TYPE IoEd12dssShutter :
STRUCT	
	OutputSwitchContactClosure	AT %Q* : BOOL;	
	
	inputShutter1 AT %I* : BOOL;
	inputShutter2 AT %I* : BOOL;
END_STRUCT
END_TYPE

(* stored: Version 1.1.0.1, ProductVersion 3.1.4024.4
   DUT IoEd12dssShutter: Id {a2021377-fd66-4d2e-89df-28c7cf5fc0ac} *)
